TYPE test :
STRUCT
END_STRUCT
END_TYPE

(* stored: Version 1.1.0.1, ProductVersion 3.1.4022.18
   DUT test: Id {8e47eb27-a1a8-4b38-93ac-ad10d0f4c9ec} *)
